(* IEC 61131-3 sources: iec-modularization/src/test/resources, 8 files *)

(* ---- bi_call_graph1.st ---- *)
FUNCTION_BLOCK FB1
END_FUNCTION_BLOCK

FUNCTION_BLOCK FB2A
VAR
	INST_FB1 : FB1;
END_VAR
	INST_FB1();
END_FUNCTION_BLOCK

FUNCTION_BLOCK FB3
VAR
	INST_FB1 : FB1;
	INST_FB2 : FB2A;
END_VAR
	INST_FB1();
	INST_FB2();
END_FUNCTION_BLOCK

(* ---- bi_call_graph2.st ---- *)
FUNCTION_BLOCK FB1
END_FUNCTION_BLOCK

FUNCTION_BLOCK FB2B
VAR
	INST_FB1 : FB1;
END_VAR
	INST_FB1();
END_FUNCTION_BLOCK

FUNCTION_BLOCK FB3
VAR
	INST_FB1 : FB1;
	INST_FB2 : FB2B;
END_VAR
	INST_FB1();
	INST_FB2();
END_FUNCTION_BLOCK

(* ---- embed_test.st ---- *)
FUNCTION_BLOCK FB
VAR_INPUT
	X : UINT;
END_VAR
VAR_OUTPUT
	Y : UINT;
END_VAR
	Y := X+1;
	Y := X+5;
	Y := X+4;
END_FUNCTION_BLOCK

FUNCTION_BLOCK PGRM
VAR
	INST_FB : FB;
END_VAR
	INST_FB.X := 5;
	INST_FB();
END_FUNCTION_BLOCK

(* ---- program1.st ---- *)
FUNCTION_BLOCK FB
VAR_INPUT
	X : UINT;
END_VAR
VAR_OUTPUT
	Y : UINT;
END_VAR
	Y := X+1;
	Y := X+5;
END_FUNCTION_BLOCK

FUNCTION_BLOCK PGRM
VAR_INPUT
	X : UINT;
END_VAR
VAR_OUTPUT
	Y : UINT;
END_VAR
VAR
	INST_FB : FB;
END_VAR
	INST_FB.X := X + 5;
	INST_FB();
	Y := INST_FB.Y;
END_FUNCTION_BLOCK

(* ---- program2.st ---- *)
FUNCTION_BLOCK FB
VAR_INPUT
	X : UINT;
END_VAR
VAR_OUTPUT
	Y : UINT;
END_VAR
	Y := X+5;
	Y := X+3;
END_FUNCTION_BLOCK

FUNCTION_BLOCK PGRM
VAR_INPUT
	X : UINT;
END_VAR
VAR_OUTPUT
	Y : UINT;
END_VAR
VAR
	INST_FB : FB;
END_VAR
	INST_FB.X := X + 7;
	INST_FB();
	Y := INST_FB.Y;
END_FUNCTION_BLOCK

(* ---- simple_call_graph.st ---- *)
FUNCTION_BLOCK FB1
END_FUNCTION_BLOCK

FUNCTION_BLOCK FB2
VAR
	INST_FB1 : FB1;
END_VAR
	INST_FB1();
END_FUNCTION_BLOCK

FUNCTION_BLOCK FB3
VAR
	INST_FB1 : FB1;
	INST_FB2 : FB2;
END_VAR
	INST_FB1();
	INST_FB2();
END_FUNCTION_BLOCK

(* ---- structural_equal1.st ---- *)
FUNCTION_BLOCK TEST_FB
VAR_INPUT
	A : INT;
	B : INT;
END_VAR
VAR_OUTPUT
	C : INT;
END_VAR
	C := A * B + B + B;
END_FUNCTION_BLOCK

(* ---- structural_equal2.st ---- *)
FUNCTION_BLOCK TEST_FB
VAR_INPUT
	A : INT;
END_VAR
VAR_INPUT
	B : INT;
END_VAR
VAR_OUTPUT
	C : INT;
END_VAR
	C := (((A * B) + B) + B);
END_FUNCTION_BLOCK
